FUNCTION_BLOCK FB_FallibleINTMock IMPLEMENTS I_FallibleINT
VAR
    bError : BOOL;
    sErrorMsg : T_MaxString;
    nVal : INT;
END_VAR


METHOD ClearError

bError := FALSE;
sErrorMsg := '';
END_METHOD


METHOD GetError : BOOL

GetError := THIS^.bError;
END_METHOD


METHOD GetErrorMsg : T_MaxString

GetErrorMsg := sErrorMsg;
END_METHOD


METHOD PUBLIC SetError
VAR_INPUT
    sMsg : T_MaxString;
END_VAR

THIS^.bError := TRUE;
END_METHOD


PROPERTY Val : INT
GET

Val := THIS^.nVal;
END_GET
SET

THIS^.nVal := Val;
END_SET
END_PROPERTY

END_FUNCTION_BLOCK

(* stored: Version 1.1.0.1
   POU FB_FallibleINTMock: Id {25a1d111-4045-47b7-859c-1db48ea9bedf}, SpecialFunc None
   Method ClearError: Id {8faf1427-6fc9-4421-8472-72fe59e69e9a}
   Method GetError: Id {e2363786-6e3d-4383-bf81-505a261a87bc}
   Method GetErrorMsg: Id {62455b1c-817d-48ca-94e0-f404c74eaab0}
   Method SetError: Id {3bc79bbf-4e63-4e94-b0ae-15a396cbc635}
   Property Val: Id {1388d4ff-d7bf-4c33-ae6d-7a137c96929d}
   Get Get: Id {e281da4e-4dc4-4aca-801f-3155e3fabfe6}
   Set Set: Id {f1c02087-ad76-4076-8c49-3337df0388b7} *)
